(* IEC 61131-3 sources: CSVFileLib/src/Ar/CSVFileLib, 5 files *)

(* ---- CSVFileLib_enum.typ ---- *)
(*
* File: CSVFileLib_enum.typ
* Copyright (c) 2023 Loupe
* https://loupe.team
*
* This file is part of CSVFileLib, licensed under the MIT License.
*
*)

TYPE
	CSV_ERR_enum :
		(
		CSV_ERR_PVITEM_ENUM := 14713,
		CSV_ERR_INVALIDINPUT := 50000,
		CSV_ERR_MEMCFG,
		CSV_ERR_MEMALLOC,
		CSV_ERR_NOTINITIALIZED,
		CSV_ERR_LINEFAILURE,
		CSV_ERR_BUFFERFULL,
		CSV_ERR_LOGNOTAVAILABLE,
		CSV_ERR_LOGFULL,
		CSV_ERR_INVALIDOPERATION,
		CSV_ERR_COMMENT,
		CSV_ERR_NOVARNAMEFOUND,
		CSV_ERR_NOVALUEFOUND,
		CSV_ERR_INVALIDVALUE,
		CSV_ERR_UNSUPPORTEDTYPE,
		CSV_ERR_INVALIDTYPE,
		CSV_ERR_MAXLEVELREACHED,
		CSV_ERR_PREFIXNOTSTRUCTURE,
		CSV_ERR_EMPTYFILENAME,
		CSV_ERR_BUSY := 65535
		);
	CSV_TYPE_enum :
		(
		CSV_TYPE_STRUCT := 0, (*0*)
		CSV_TYPE_BOOL,
		CSV_TYPE_SINT,
		CSV_TYPE_INT,
		CSV_TYPE_DINT,
		CSV_TYPE_USINT, (*5*)
		CSV_TYPE_UINT,
		CSV_TYPE_UDINT,
		CSV_TYPE_REAL,
		CSV_TYPE_STRING,
		CSV_TYPE_ULINT, (*10*)
		CSV_TYPE_DATE_AND_TIME,
		CSV_TYPE_TIME,
		CSV_TYPE_DATE,
		CSV_TYPE_LREAL,
		CSV_TYPE_ARRAY_OF_STRUCT, (*15*)
		CSV_TYPE_TIME_OF_DAY,
		CSV_TYPE_BYTE,
		CSV_TYPE_WORD,
		CSV_TYPE_DWORD,
		CSV_TYPE_LWORD, (*20*)
		CSV_TYPE_WSTRING, (*21*)
		CSV_TYPE_LINT := 23 (*23*)
		);
	CSV_BITFORMAT_enum :
		(
		CSV_BITFORMAT_HEX_0X := 0, (*0x00FF - default*)
		CSV_BITFORMAT_HEX_IEC, (*16#00FF*)
		CSV_BITFORMAT_DECIMAL (*255*)
		);
	CSV_INFO_enum :
		(
		CSV_INFO_NOVARNAMEFOUND, (*0*)
		CSV_INFO_NOVALUEFOUND,
		CSV_INFO_ADDRESSNOTFOUND,
		CSV_INFO_DATATYPENOTFOUND,
		CSV_INFO_INVALIDVALUE,
		CSV_INFO_UNSUPPORTEDTYPE, (*5*)
		CSV_INFO_INVALIDTYPE,
		CSV_INFO_INVALIDINPUT,
		CSV_INFO_FILEFULL,
		CSV_INFO_INFONOTFOUND,
		CSV_INFO_MAXLEVELREACHED, (*10*)
		CSV_INFO_ITEMNOTFOUND,
		CSV_INFO_PREFIXNOTSTRUCTURE,
		CSV_INFO_VERBOSE_VARNAME,
		CSV_INFO_VERBOSE_VALUE,
		CSV_INFO_VERBOSE_DESCRIPTION, (*15*)
		CSV_INFO_VERBOSE_VARADDRESS,
		CSV_INFO_VERBOSE_VARTYPE,
		CSV_INFO_VERBOSE_VARLENGTH,
		CSV_INFO_VERBOSE_VARDIMENSION,
		CSV_INFO_VERBOSE_COMMENT, (*20*)
		CSV_INFO_DONE (*21*)
		);
	CSV_FILELIST_ST_enum :
		(
		CSV_FILELIST_ST_IDLE,
		CSV_FILELIST_ST_DIRINFO,
		CSV_FILELIST_ST_DIRREAD,
		CSV_FILELIST_ST_
		);
	CSV_ST_enum :
		(
		CSV_ST_IDLE := 0, (*0*)
		CSV_ST_GET_TEMPLATE,
		CSV_ST_EXPANDVARS,
		CSV_ST_OPEN,
		CSV_ST_PROCESS,
		CSV_ST_DELETELOG,
		CSV_ST_SAVELOG, (*4*)
		CSV_ST_CURRENTOPERATION,
		CSV_ST_DELETETEMP := 100, (*100*)
		CSV_ST_SAVETEMP,
		CSV_ST_DELETEORIGINAL,
		CSV_ST_RENAMETEMP, (*103*)
		CSV_ST_DELETEFILE := 200, (*200*)
		CSV_ST_ERROR := 999 (*999*)
		);
	CSV_OP_enum :
		(
		CSV_OP_INVALID := 0,
		CSV_OP_OPEN,
		CSV_OP_SAVE,
		CSV_OP_DELETE
		);
END_TYPE

(* ---- CSVFileMgr.typ ---- *)
(*
* File: CSVFileMgr.typ
* Copyright (c) 2023 Loupe
* https://loupe.team
*
* This file is part of CSVFileLib, licensed under the MIT License.
*
*)

TYPE
	CSVFileVariable_typ : 	STRUCT
		Name : STRING[CSV_STRLEN_VARNAME];
		Value : STRING[CSV_STRLEN_VARVALUE];
		Description : STRING[CSV_STRLEN_VARDESCRIPTION];
		Address : UDINT;
		DataType : UDINT;
		Length : UDINT;
		Dimension : UINT;
	END_STRUCT;
	CSVFileMgr_StructLevel_typ : 	STRUCT
		Name : STRING[CSV_STRLEN_VARNAME];
		DataType : UDINT;
		Length : UDINT;
		Dimension : UINT;
		iItem : UINT;
	END_STRUCT;
	CSVFileMgr_StructData_typ : 	STRUCT
		iLevel : INT;
		Level : ARRAY[0..CSV_MAI_LEVEL]OF CSVFileMgr_StructLevel_typ;
	END_STRUCT;
	CSVFileMgr_Int_Buffer_typ : 	STRUCT
		pData : UDINT;
		CurrentLength : UDINT;
		MaxLength : UDINT;
	END_STRUCT;
	CSVFileMgr_Internal_typ : 	STRUCT
		Initialized : BOOL;
		CurrOperation : DINT;
		ProcessStatus : UINT;
		ExpandStatus : UINT;
		ExpandError : BOOL;
		ReadBuffer : CSVFileMgr_Int_Buffer_typ;
		WriteBuffer : CSVFileMgr_Int_Buffer_typ;
		LogBuffer : CSVFileMgr_Int_Buffer_typ;
		pLine : UDINT;
		LineNumber : UDINT;
		pToken : UDINT;
		pString : UDINT;
		pReentry : UDINT;
		SuccessfulLineCount : UDINT;
		FailedLineCount : UDINT;
		ScanCount : UDINT;
		StructureData : CSVFileMgr_StructData_typ;
		iVar : USINT;
		FileRename : FileRename;
		FIOWrap : FIOWrap_typ;
		CMD : CSVFileMgr_IN_CMD_typ;
		TempFileName : STRING[CSV_STRLEN_TEMPFILENAME];
		TemplateVariable : CSVFileVariable_typ;
		pUserVariable : UDINT;
		StartState : DINT;
	END_STRUCT;
	CSVFileMgr_OUT_STAT_typ : 	STRUCT
		Busy : BOOL;
		Done : BOOL;
		Error : BOOL;
		ErrorID : UINT;
		ErrorString : STRING[CSV_STRLEN_ERROR];
		ErrorLevel : USINT;
		ErrorState : DINT;
		State : DINT;
	END_STRUCT;
	CSVFileMgr_OUT_typ : 	STRUCT
		STAT : CSVFileMgr_OUT_STAT_typ;
	END_STRUCT;
	CSVFileMgr_IN_CFG_typ : 	STRUCT
		MaxFileSize : UDINT;
		MaxLineLength : UDINT;
		MaxLinesPerScan : UDINT;
		VerboseLog : BOOL;
		LogFileName : STRING[CSV_STRLEN_FILENAME];
		DisableLogging : BOOL;
		LoggerName : STRING[LOG_STRLEN_LOGGERNAME];
		DoubleSigFigs : USINT;
		BitStringFormat : USINT; (*How BYTE/WORD/DWORD values are written, see CSV_BITFORMAT_enum. Reading accepts hex and decimal regardless of this setting*)
	END_STRUCT;
	CSVFileMgr_IN_PAR_typ : 	STRUCT
		FileDevice : STRING[CSV_STRLEN_FILEDEVICE];
		FileName : STRING[CSV_STRLEN_FILENAME];
		VariableList : ARRAY[0..CSV_MAI_VARLIST]OF STRING[CSV_STRLEN_VARNAME];
		Prefix : STRING[CSV_STRLEN_VARNAME];
		pUserVariable : UDINT;
	END_STRUCT;
	CSVFileMgr_IN_CMD_typ : 	STRUCT
		OpenFile : BOOL;
		UpdateFile : BOOL;
		SaveVariableListToFile : BOOL;
		DeleteFile : BOOL;
		AcknowledgeError : BOOL;
	END_STRUCT;
	CSVFileMgr_IN_typ : 	STRUCT
		CMD : CSVFileMgr_IN_CMD_typ;
		PAR : CSVFileMgr_IN_PAR_typ;
		CFG : CSVFileMgr_IN_CFG_typ;
	END_STRUCT;
	CSVFileMgr_typ : 	STRUCT
		IN : CSVFileMgr_IN_typ;
		OUT : CSVFileMgr_OUT_typ;
		Internal : CSVFileMgr_Internal_typ;
	END_STRUCT;
END_TYPE

(* ---- CSVFileMgr_HMI.typ ---- *)
(*
* File: CSVFileMgr_HMI.typ
* Copyright (c) 2023 Loupe
* https://loupe.team
*
* This file is part of CSVFileLib, licensed under the MIT License.
*
*)

TYPE
	CSVFileMgr_HMI_Internal_typ : 	STRUCT
		ProgressTimer : TON_10ms;
		HMI_CMD_Active : BOOL;
		HMI_CMD_Active_Old : BOOL;
	END_STRUCT;
	CSVFileMgr_HMI_TextSnippets_typ : 	STRUCT
		FileName : STRING[CSV_STRLEN_FILENAME];
		PopupHeader : STRING[CSV_STRLEN_FILENAME];
		Action : STRING[CSV_STRLEN_FILENAME];
		ProgressLabel : STRING[CSV_STRLEN_FILENAME];
		ErrorID : UINT;
		ErrorString : STRING[CSV_STRLEN_ERROR];
	END_STRUCT;
	CSVFileMgr_HMI_ErrorStatus_typ : 	STRUCT
		StatusDP : UINT;
		AcknowledgeError : HMI_Button_typ;
	END_STRUCT;
	CSVFileMgr_HMI_Progress_typ : 	STRUCT
		StatusDP : UINT;
		Progress : UDINT;
	END_STRUCT;
	CSVFileMgr_HMI_DeleteConfirm_typ : 	STRUCT
		StatusDP : UINT;
		Yes : HMI_Button_typ;
		No : HMI_Button_typ;
	END_STRUCT;
	CSVFileMgr_HMI_DialogBox_typ : 	STRUCT
		StatusDP : UINT;
		FileNameList : ARRAY[0..CSV_MAI_FILELIST]OF STRING[LIST_BOX_STRING_SIZE];
		FileBrowser : HMIFileBrowse;
		PageUp : HMI_Button_typ;
		PageDown : HMI_Button_typ;
		Action : HMI_Button_typ;
		Cancel : HMI_Button_typ;
	END_STRUCT;
	CSVFileMgr_HMI_Main_typ : 	STRUCT
		OpenFile : HMI_Button_typ;
		UpdateFile : HMI_Button_typ;
		SaveVariableListToFile : HMI_Button_typ;
		DeleteFile : HMI_Button_typ;
	END_STRUCT;
	CSVFileMgr_HMI_typ : 	STRUCT
		Main : CSVFileMgr_HMI_Main_typ;
		DialogBox : CSVFileMgr_HMI_DialogBox_typ;
		DeleteConfirm : CSVFileMgr_HMI_DeleteConfirm_typ;
		Progress : CSVFileMgr_HMI_Progress_typ;
		ErrorStatus : CSVFileMgr_HMI_ErrorStatus_typ;
		TextSnippets : CSVFileMgr_HMI_TextSnippets_typ;
		Internal : CSVFileMgr_HMI_Internal_typ;
	END_STRUCT;
END_TYPE

(* ---- CSVFileLib.fun ---- *)
(*
* File: CSVFileLib.fun
* Copyright (c) 2023 Loupe
* https://loupe.team
*
* This file is part of CSVFileLib, licensed under the MIT License.
*
*)

FUNCTION CSVFn_Init : UINT (*CSVFileMgr initialization function*)
	VAR_IN_OUT
		t : CSVFileMgr_typ;
	END_VAR
END_FUNCTION

FUNCTION CSVOpenFile_Init : UINT (*Open a file in an INIT routine*)
	VAR_IN_OUT
		t : CSVFileMgr_typ;
	END_VAR
END_FUNCTION

FUNCTION CSVFn_Cyclic : UINT (*CSVFileMgr cyclic function*)
	VAR_IN_OUT
		t : CSVFileMgr_typ;
	END_VAR
END_FUNCTION

FUNCTION csvInitBuffer : UINT (*Initialize a buffer*)
	VAR_INPUT
		BufferLength : UDINT;
	END_VAR
	VAR_IN_OUT
		pBuffer : CSVFileMgr_Int_Buffer_typ;
	END_VAR
END_FUNCTION

FUNCTION csvClearBuffer : UINT (*Clear a buffer*)
	VAR_IN_OUT
		pBuffer : CSVFileMgr_Int_Buffer_typ;
	END_VAR
END_FUNCTION

FUNCTION csvAddToBuffer : UINT (*Add data to the end of a buffer, checking for overflow*)
	VAR_INPUT
		pData : UDINT;
		DataLength : UDINT;
	END_VAR
	VAR_IN_OUT
		pBuffer : CSVFileMgr_Int_Buffer_typ;
	END_VAR
END_FUNCTION

FUNCTION csvSetError : UINT (*Set error status on CSVFileMgr*)
	VAR_INPUT
		ErrorID : UINT;
	END_VAR
	VAR_IN_OUT
		t : CSVFileMgr_typ;
	END_VAR
END_FUNCTION

FUNCTION csvExpandVar : UINT (*Expand a complex variable into simple variables*)
	VAR_INPUT
		pVarName : UDINT;
	END_VAR
	VAR_IN_OUT
		pBuffer : CSVFileMgr_Int_Buffer_typ;
		pStructData : CSVFileMgr_StructData_typ;
		t : CSVFileMgr_typ;
	END_VAR
END_FUNCTION

FUNCTION csvProcessData : UINT (*Process data from file*)
	VAR_IN_OUT
		t : CSVFileMgr_typ;
	END_VAR
END_FUNCTION

FUNCTION csvAddLogInfo : UINT (*Add information to the parse status log*)
	VAR_INPUT
		InfoID : UINT;
		LineNumber : UDINT;
		pAddInfo : UDINT;
	END_VAR
	VAR_IN_OUT
		t : CSVFileMgr_typ;
	END_VAR
END_FUNCTION

FUNCTION csvParseLine : UINT (*Parse one line of the file*)
	VAR_INPUT
		pLine : UDINT;
		LineNumber : UDINT;
	END_VAR
	VAR_IN_OUT
		pVariable : CSVFileVariable_typ;
		t : CSVFileMgr_typ;
	END_VAR
END_FUNCTION

FUNCTION csvGetVarInfo : UINT (*Get variable address and data type based on variable name*)
	VAR_INPUT
		LineNumber : UDINT;
	END_VAR
	VAR_IN_OUT
		pVariable : CSVFileVariable_typ;
		t : CSVFileMgr_typ;
	END_VAR
END_FUNCTION

FUNCTION csvOpenVar : UINT (*Process one variable of an Open operation*)
	VAR_INPUT
		LineNumber : UDINT;
	END_VAR
	VAR_IN_OUT
		pVariable : CSVFileVariable_typ;
		t : CSVFileMgr_typ;
	END_VAR
END_FUNCTION

FUNCTION csvSaveVar : UINT (*Process one variable of a Save operation*)
	VAR_INPUT
		LineNumber : UDINT;
	END_VAR
	VAR_IN_OUT
		pVariable : CSVFileVariable_typ;
		t : CSVFileMgr_typ;
	END_VAR
END_FUNCTION

FUNCTION csvWriteHeader : UINT (*Write the header to the file*)
	VAR_IN_OUT
		t : CSVFileMgr_typ;
	END_VAR
END_FUNCTION

FUNCTION csvRemovePrefix : UINT (*Remove the prefix from the string if necessary*)
	VAR_INPUT
		MaxLength : UDINT;
	END_VAR
	VAR_IN_OUT
		String : STRING[1];
		Prefix : STRING[1];
	END_VAR
END_FUNCTION

FUNCTION csvAddPrefix : UINT (*Add a prefix to a string, unconditionally*)
	VAR_INPUT
		MaxLength : UDINT;
	END_VAR
	VAR_IN_OUT
		String : STRING[1];
		Prefix : STRING[1];
	END_VAR
END_FUNCTION

FUNCTION CSVFn_HMI_Cyclic : UINT (*CSVFileMgr cyclic HMI function*)
	VAR_IN_OUT
		HMI : CSVFileMgr_HMI_typ;
		t : CSVFileMgr_typ;
	END_VAR
END_FUNCTION

FUNCTION csvhmiGenerateFileListString : UINT (*Generate the file list string for a given file*)
	VAR_INPUT
		pFileListString : UDINT;
	END_VAR
	VAR_IN_OUT
		pDirReadData : fiDIR_READ_DATA;
	END_VAR
END_FUNCTION

FUNCTION csvDTOA : UDINT (*Convert double to string*)
	VAR_INPUT
		value : LREAL;
		pString : UDINT;
		numSigFigs : USINT;
	END_VAR
END_FUNCTION

(* ---- CSVFileLib.var ---- *)
(*
* File: CSVFileLib.var
* Copyright (c) 2023 Loupe
* https://loupe.team
*
* This file is part of CSVFileLib, licensed under the MIT License.
*
*)
VAR CONSTANT
	CSV_PADDINGCHARS : STRING[6] := ' $T$R$L$P$"';
END_VAR
(*Max Array Indices*)
VAR CONSTANT
	CSV_MAI_LEVEL : USINT := 29;
	CSV_MAI_VARLIST : USINT := 99;
	CSV_MAI_FILELIST : UINT := 299;
END_VAR
(*String Lengths*)
VAR CONSTANT
	CSV_STRLEN_FILENAME : UINT := 260;
	CSV_STRLEN_TEMPFILENAME : UINT := CSV_STRLEN_FILENAME + 3;
	CSV_STRLEN_FILEDEVICE : UINT := 260;
	CSV_STRLEN_FILENAMEDISPLAY : USINT := 30;
	CSV_STRLEN_MINSPACING : USINT := 4;
	CSV_STRLEN_TIMESTAMP : USINT := 16;
	CSV_STRLEN_ERROR : USINT := 99;
	CSV_STRLEN_VARNAME : USINT := 120;
	CSV_STRLEN_VARVALUE : UINT := 500;
	CSV_STRLEN_VARDESCRIPTION : USINT := 120;
	CSV_STRLEN_FILELIST : USINT := CSV_STRLEN_FILENAMEDISPLAY + CSV_STRLEN_MINSPACING + CSV_STRLEN_TIMESTAMP;
	CSV_STRLEN_INFOSTRING : USINT := 200;
	CSV_STRLEN_HEADER : UINT := 44+320;
END_VAR
(*Default CFG values*)
VAR CONSTANT
	CSV_DEFAULT_MAXFILESIZE : UDINT := 65536;
	CSV_DEFAULT_MAXLINELENGTH : UDINT := 500;
	CSV_DEFAULT_MAXLINESPERSCAN : UDINT := 500;
	CSV_DEFAULT_LOGGERNAME : STRING[LOG_STRLEN_LOGGERNAME] := 'Files';
	CSV_DEFAULT_SIGFIGS : USINT := 16;
END_VAR
(*Data type limits*)
VAR CONSTANT
	CSV_MIN_SINT : DINT := -128;
	CSV_MAX_SINT : DINT := 127;
	CSV_MIN_INT : DINT := -32768;
	CSV_MAX_INT : DINT := 32767;
	CSV_MIN_DINT : DINT := -2147483647;
	CSV_MAX_DINT : DINT := 2147483647;
	CSV_MIN_USINT : DINT := 0;
	CSV_MAX_USINT : DINT := 255;
	CSV_MIN_UINT : DINT := 0;
	CSV_MAX_UINT : DINT := 65535;
	CSV_MIN_UDINT : UDINT := 0;
	CSV_MAX_UDINT : UDINT := 4294967295;
	CSV_MAX_BYTE : UDINT := 255;
	CSV_MAX_WORD : UDINT := 65535;
	CSV_MAX_DWORD : UDINT := 4294967295;
	CSV_MIN_REAL : REAL := -3.4E038;
	CSV_MAX_REAL : REAL := 3.4E038;
	CSV_MIN_LREAL : LREAL := -1.7976931348623158E308;
	CSV_MAX_LREAL : LREAL := 1.7976931348623158E308;
END_VAR
